FUNCTION_BLOCK EBM_Speed
VAR_INPUT
	EN: BOOL;
	ModbusRTU: REFERENCE TO ModbusRTU;
	Address: BYTE := 101;
END_VAR
VAR_OUTPUT
	ENO: BOOL;
	Speed: LREAL;
END_VAR
VAR
	ModbusWord_T_ActualSpeed: ModbusReadWord;
	ModbusWord_T_nMax: ModbusReadWord;
	ActualSpeed: LREAL;
END_VAR
VAR // added by the converter: edge detectors and wires of the graphical bodies
    _w1 : ANY;
    _w2 : LREAL;
    _w3 : INT;
END_VAR

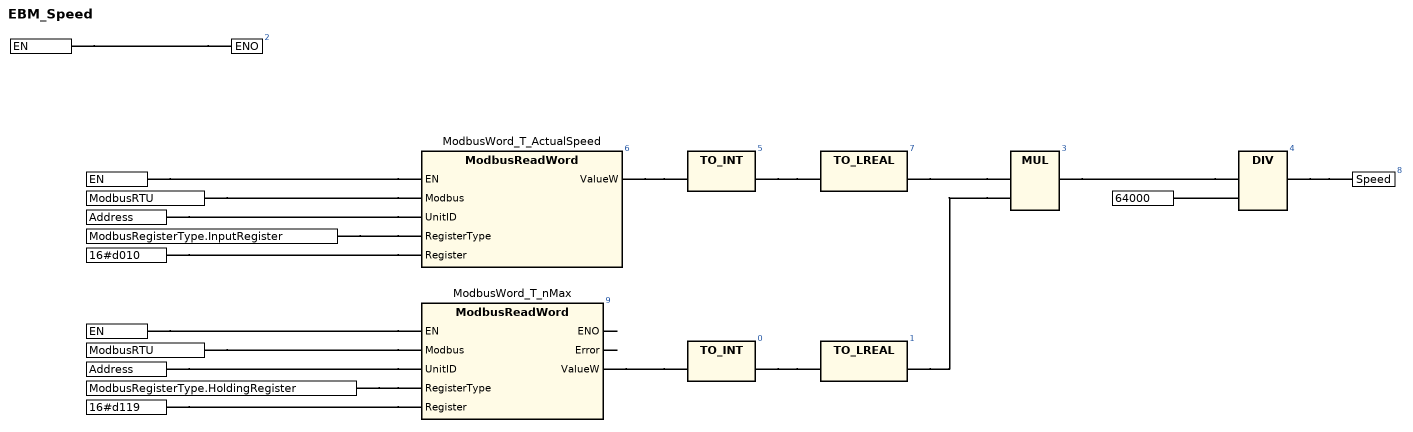
ENO := EN;
_w2 := (_w1 * TO_LREAL(TO_INT(ModbusWord_T_nMax.ValueW))) / 64000;
_w3 := TO_INT(ModbusWord_T_ActualSpeed.ValueW);
ModbusWord_T_ActualSpeed(
    EN := EN,
    Modbus := ModbusRTU,
    UnitID := Address,
    RegisterType := ModbusRegisterType.InputRegister,
    Register := 16#d010); // ModbusReadWord
_w1 := TO_LREAL(_w3);
Speed := _w2;
ModbusWord_T_nMax(
    EN := EN,
    Modbus := ModbusRTU,
    UnitID := Address,
    RegisterType := ModbusRegisterType.HoldingRegister,
    Register := 16#d119); // ModbusReadWord

END_FUNCTION_BLOCK

(* stored: Version 1.1.0.1, ProductVersion 3.1.4024.6
   POU EBM_Speed: Id {142fc662-e25d-44b2-8959-18bb820406b2}, SpecialFunc None *)
